{attribute 'enable_dynamic_creation'}
FUNCTION_BLOCK Snapshot
VAR
	pEditor : POINTER TO RecipeEditor;
	sTitle : STRING;
	sRecipeSteps : ARRAY[1..5] OF STRING;
END_VAR

METHOD FB_exit : BOOL
VAR_INPUT
	bInCopyCode : BOOL; // if TRUE, the exit method is called for exiting an instance that is copied afterwards (online change).
END_VAR
// Clear the pointer on exit
IF pEditor <> 16#0000 THEN
	pEditor := 16#0000;
END_IF
END_METHOD

METHOD FB_init : BOOL
VAR_INPUT
	bInitRetains : BOOL; // if TRUE, the retain variables are initialized (warm start / cold start)
	bInCopyCode : BOOL;  // if TRUE, the instance afterwards gets moved into the copy code (online change)
	pEditor : POINTER TO RecipeEditor;
	sTitle : STRING;
	sRecipeSteps : ARRAY[1..5] OF STRING;
END_VAR
THIS^.pEditor := pEditor;
THIS^.sTitle := sTitle;
THIS^.sRecipeSteps := sRecipeSteps;
END_METHOD

METHOD restore
VAR_INPUT
END_VAR
pEditor^.setTitle(THIS^.sTitle);
pEditor^.setRecipe(THIS^.sRecipeSteps);
ADSLOGSTR( msgCtrlMask := ADSLOG_MSGTYPE_LOG, msgFmtStr := 'PLC Msg.: %s', strArg := 'Snapshot restored...');
END_METHOD

END_FUNCTION_BLOCK

(* stored: Version 1.1.0.1, ProductVersion 3.1.4024.12
   POU Snapshot: Id {14f1b39a-6b83-4b3d-8c16-e8df624b3a28}, SpecialFunc None
   Method FB_exit: Id {6dcc51a9-78b0-448b-8b92-b57f979dcb32}
   Method FB_init: Id {06c666fa-9174-47c9-8d0d-ce8b18b1188d}
   Method restore: Id {788b526b-1fd4-44a0-9ef2-d3ab3a33bd5f} *)
